PROGRAM SP1_2_Y111
VAR
	CompareOutput111_00: CMP_OC_DW;
	CompareOutput111_01: CMP_OC_DW;
	CompareOutput111_02: CMP_OC_DW;
	CompareOutput111_03: CMP_OC_DW;
	CompareOutput111_04: CMP_OC_DW;
	CompareOutput111_05: CMP_OC_DW;
	CompareOutput111_06: CMP_OC_DW;
	CompareOutput111_07: CMP_OC_DW;
	CompareOutput111_08: CMP_OC_DW;
	CompareOutput111_09: CMP_OC_DW;
	CompareOutput111_10: CMP_OC_DW;
	CompareOutput111_11: CMP_OC_DW;
	CompareOutput111_12: CMP_OC_DW;
	CompareOutput111_13: CMP_OC_DW;
	CompareOutput111_14: CMP_OC_DW;
	CompareOutput111_15: CMP_OC_DW;

END_VAR

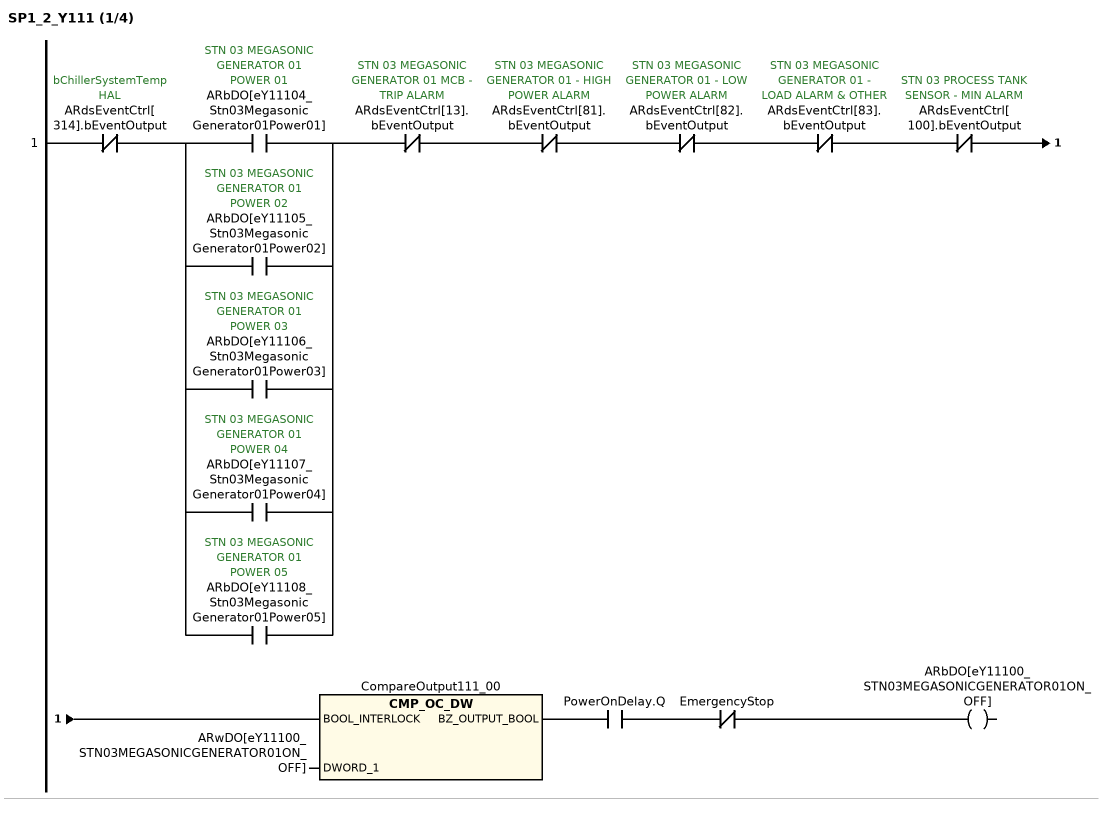
// NETWORK 1
//   ARdsEventCtrl[314].bEventOutput: bChillerSystemTempHAL
//   ARbDO[eY11104_Stn03MegasonicGenerator01Power01]: STN 03 MEGASONIC GENERATOR 01 POWER 01
//   ARbDO[eY11105_Stn03MegasonicGenerator01Power02]: STN 03 MEGASONIC GENERATOR 01 POWER 02
//   ARbDO[eY11106_Stn03MegasonicGenerator01Power03]: STN 03 MEGASONIC GENERATOR 01 POWER 03
//   ARbDO[eY11107_Stn03MegasonicGenerator01Power04]: STN 03 MEGASONIC GENERATOR 01 POWER 04
//   ARbDO[eY11108_Stn03MegasonicGenerator01Power05]: STN 03 MEGASONIC GENERATOR 01 POWER 05
//   ARdsEventCtrl[13].bEventOutput: STN 03 MEGASONIC GENERATOR 01 MCB - TRIP ALARM
//   ARdsEventCtrl[81].bEventOutput: STN 03 MEGASONIC GENERATOR 01 - HIGH POWER ALARM
//   ARdsEventCtrl[82].bEventOutput: STN 03 MEGASONIC GENERATOR 01 - LOW POWER ALARM
//   ARdsEventCtrl[83].bEventOutput: STN 03 MEGASONIC GENERATOR 01 - LOAD ALARM & OTHER
//   ARdsEventCtrl[100].bEventOutput: STN 03 PROCESS TANK SENSOR - MIN ALARM
CompareOutput111_00(BOOL_INTERLOCK := NOT ARdsEventCtrl[314].bEventOutput AND (ARbDO[eY11104_Stn03MegasonicGenerator01Power01] OR ARbDO[eY11105_Stn03MegasonicGenerator01Power02] OR ARbDO[eY11106_Stn03MegasonicGenerator01Power03] OR ARbDO[eY11107_Stn03MegasonicGenerator01Power04] OR ARbDO[eY11108_Stn03MegasonicGenerator01Power05]) AND NOT ARdsEventCtrl[13].bEventOutput AND NOT ARdsEventCtrl[81].bEventOutput AND NOT ARdsEventCtrl[82].bEventOutput AND NOT ARdsEventCtrl[83].bEventOutput AND NOT ARdsEventCtrl[100].bEventOutput, DWORD_1 := ARwDO[eY11100_STN03MEGASONICGENERATOR01ON_OFF]); // CMP_OC_DW
ARbDO[eY11100_STN03MEGASONICGENERATOR01ON_OFF] := CompareOutput111_00.BZ_OUTPUT_BOOL AND PowerOnDelay.Q AND NOT EmergencyStop;

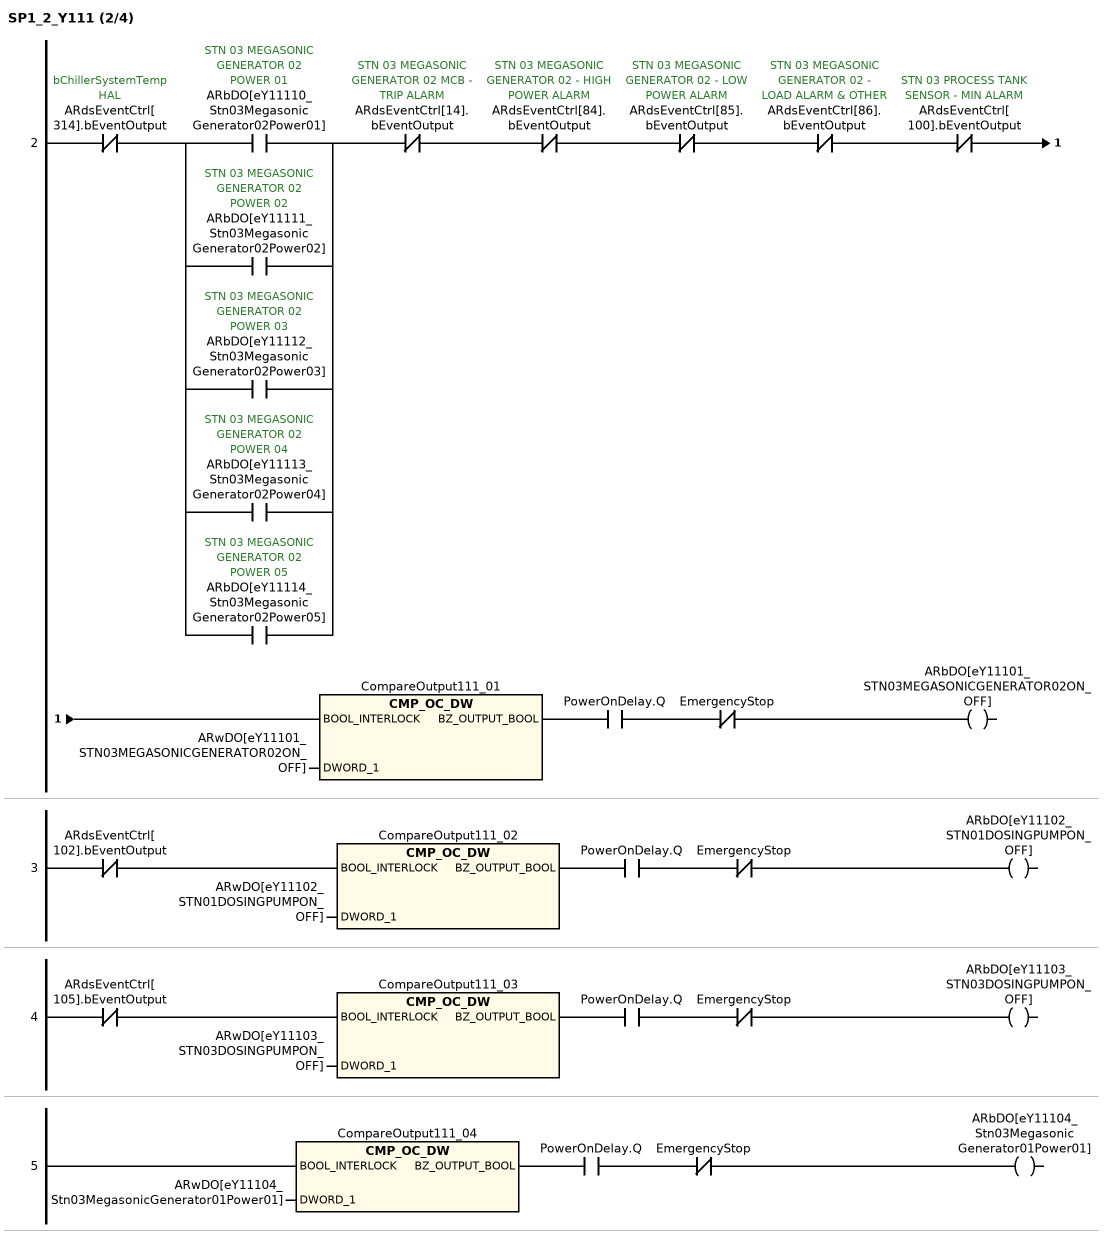
// NETWORK 2
//   ARdsEventCtrl[314].bEventOutput: bChillerSystemTempHAL
//   ARbDO[eY11110_Stn03MegasonicGenerator02Power01]: STN 03 MEGASONIC GENERATOR 02 POWER 01
//   ARbDO[eY11111_Stn03MegasonicGenerator02Power02]: STN 03 MEGASONIC GENERATOR 02 POWER 02
//   ARbDO[eY11112_Stn03MegasonicGenerator02Power03]: STN 03 MEGASONIC GENERATOR 02 POWER 03
//   ARbDO[eY11113_Stn03MegasonicGenerator02Power04]: STN 03 MEGASONIC GENERATOR 02 POWER 04
//   ARbDO[eY11114_Stn03MegasonicGenerator02Power05]: STN 03 MEGASONIC GENERATOR 02 POWER 05
//   ARdsEventCtrl[14].bEventOutput: STN 03 MEGASONIC GENERATOR 02 MCB - TRIP ALARM
//   ARdsEventCtrl[84].bEventOutput: STN 03 MEGASONIC GENERATOR 02 - HIGH POWER ALARM
//   ARdsEventCtrl[85].bEventOutput: STN 03 MEGASONIC GENERATOR 02 - LOW POWER ALARM
//   ARdsEventCtrl[86].bEventOutput: STN 03 MEGASONIC GENERATOR 02 - LOAD ALARM & OTHER
//   ARdsEventCtrl[100].bEventOutput: STN 03 PROCESS TANK SENSOR - MIN ALARM
CompareOutput111_01(BOOL_INTERLOCK := NOT ARdsEventCtrl[314].bEventOutput AND (ARbDO[eY11110_Stn03MegasonicGenerator02Power01] OR ARbDO[eY11111_Stn03MegasonicGenerator02Power02] OR ARbDO[eY11112_Stn03MegasonicGenerator02Power03] OR ARbDO[eY11113_Stn03MegasonicGenerator02Power04] OR ARbDO[eY11114_Stn03MegasonicGenerator02Power05]) AND NOT ARdsEventCtrl[14].bEventOutput AND NOT ARdsEventCtrl[84].bEventOutput AND NOT ARdsEventCtrl[85].bEventOutput AND NOT ARdsEventCtrl[86].bEventOutput AND NOT ARdsEventCtrl[100].bEventOutput, DWORD_1 := ARwDO[eY11101_STN03MEGASONICGENERATOR02ON_OFF]); // CMP_OC_DW
ARbDO[eY11101_STN03MEGASONICGENERATOR02ON_OFF] := CompareOutput111_01.BZ_OUTPUT_BOOL AND PowerOnDelay.Q AND NOT EmergencyStop;

// NETWORK 3
CompareOutput111_02(BOOL_INTERLOCK := NOT ARdsEventCtrl[102].bEventOutput, DWORD_1 := ARwDO[eY11102_STN01DOSINGPUMPON_OFF]); // CMP_OC_DW
ARbDO[eY11102_STN01DOSINGPUMPON_OFF] := CompareOutput111_02.BZ_OUTPUT_BOOL AND PowerOnDelay.Q AND NOT EmergencyStop;

// NETWORK 4
CompareOutput111_03(BOOL_INTERLOCK := NOT ARdsEventCtrl[105].bEventOutput, DWORD_1 := ARwDO[eY11103_STN03DOSINGPUMPON_OFF]); // CMP_OC_DW
ARbDO[eY11103_STN03DOSINGPUMPON_OFF] := CompareOutput111_03.BZ_OUTPUT_BOOL AND PowerOnDelay.Q AND NOT EmergencyStop;

// NETWORK 5
CompareOutput111_04(BOOL_INTERLOCK := TRUE, DWORD_1 := ARwDO[eY11104_Stn03MegasonicGenerator01Power01]); // CMP_OC_DW
ARbDO[eY11104_Stn03MegasonicGenerator01Power01] := CompareOutput111_04.BZ_OUTPUT_BOOL AND PowerOnDelay.Q AND NOT EmergencyStop;

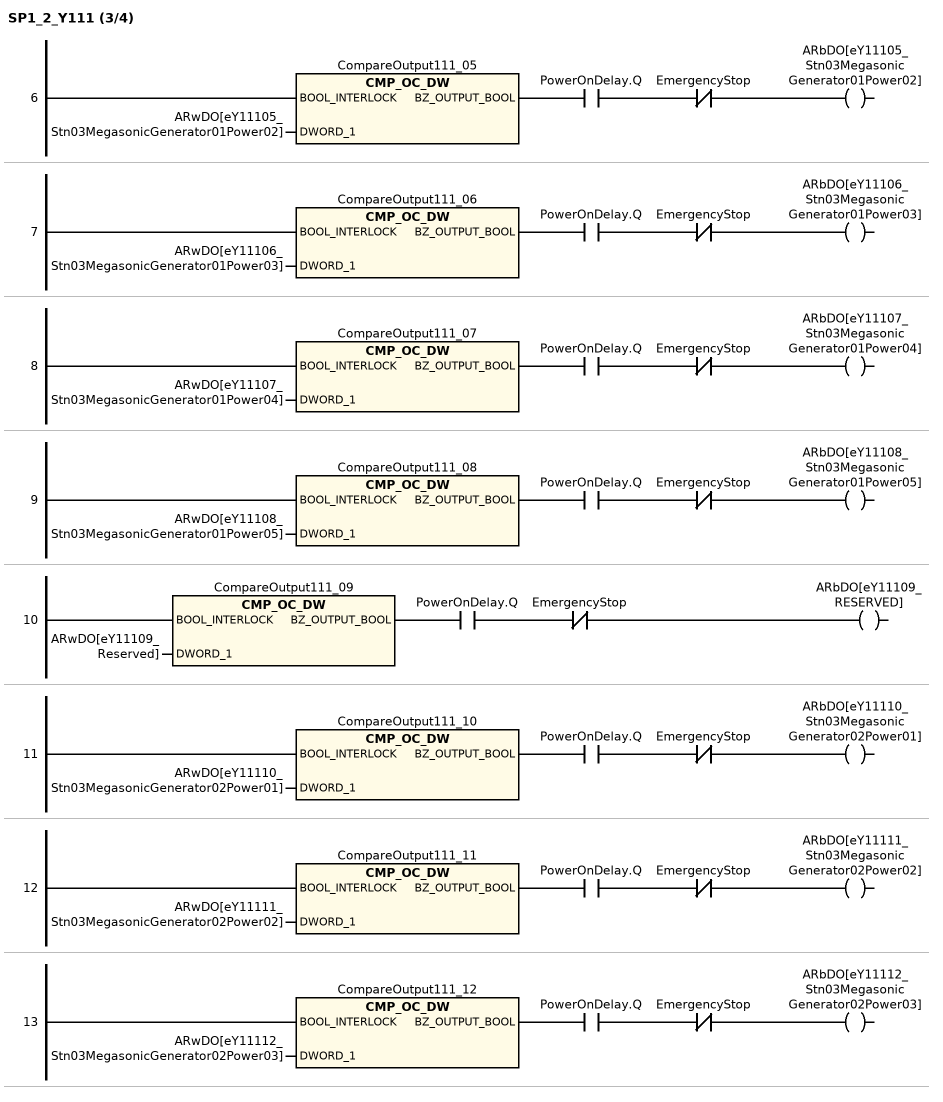
// NETWORK 6
CompareOutput111_05(BOOL_INTERLOCK := TRUE, DWORD_1 := ARwDO[eY11105_Stn03MegasonicGenerator01Power02]); // CMP_OC_DW
ARbDO[eY11105_Stn03MegasonicGenerator01Power02] := CompareOutput111_05.BZ_OUTPUT_BOOL AND PowerOnDelay.Q AND NOT EmergencyStop;

// NETWORK 7
CompareOutput111_06(BOOL_INTERLOCK := TRUE, DWORD_1 := ARwDO[eY11106_Stn03MegasonicGenerator01Power03]); // CMP_OC_DW
ARbDO[eY11106_Stn03MegasonicGenerator01Power03] := CompareOutput111_06.BZ_OUTPUT_BOOL AND PowerOnDelay.Q AND NOT EmergencyStop;

// NETWORK 8
CompareOutput111_07(BOOL_INTERLOCK := TRUE, DWORD_1 := ARwDO[eY11107_Stn03MegasonicGenerator01Power04]); // CMP_OC_DW
ARbDO[eY11107_Stn03MegasonicGenerator01Power04] := CompareOutput111_07.BZ_OUTPUT_BOOL AND PowerOnDelay.Q AND NOT EmergencyStop;

// NETWORK 9
CompareOutput111_08(BOOL_INTERLOCK := TRUE, DWORD_1 := ARwDO[eY11108_Stn03MegasonicGenerator01Power05]); // CMP_OC_DW
ARbDO[eY11108_Stn03MegasonicGenerator01Power05] := CompareOutput111_08.BZ_OUTPUT_BOOL AND PowerOnDelay.Q AND NOT EmergencyStop;

// NETWORK 10
CompareOutput111_09(BOOL_INTERLOCK := TRUE, DWORD_1 := ARwDO[eY11109_Reserved]); // CMP_OC_DW
ARbDO[eY11109_RESERVED] := CompareOutput111_09.BZ_OUTPUT_BOOL AND PowerOnDelay.Q AND NOT EmergencyStop;

// NETWORK 11
CompareOutput111_10(BOOL_INTERLOCK := TRUE, DWORD_1 := ARwDO[eY11110_Stn03MegasonicGenerator02Power01]); // CMP_OC_DW
ARbDO[eY11110_Stn03MegasonicGenerator02Power01] := CompareOutput111_10.BZ_OUTPUT_BOOL AND PowerOnDelay.Q AND NOT EmergencyStop;

// NETWORK 12
CompareOutput111_11(BOOL_INTERLOCK := TRUE, DWORD_1 := ARwDO[eY11111_Stn03MegasonicGenerator02Power02]); // CMP_OC_DW
ARbDO[eY11111_Stn03MegasonicGenerator02Power02] := CompareOutput111_11.BZ_OUTPUT_BOOL AND PowerOnDelay.Q AND NOT EmergencyStop;

// NETWORK 13
CompareOutput111_12(BOOL_INTERLOCK := TRUE, DWORD_1 := ARwDO[eY11112_Stn03MegasonicGenerator02Power03]); // CMP_OC_DW
ARbDO[eY11112_Stn03MegasonicGenerator02Power03] := CompareOutput111_12.BZ_OUTPUT_BOOL AND PowerOnDelay.Q AND NOT EmergencyStop;

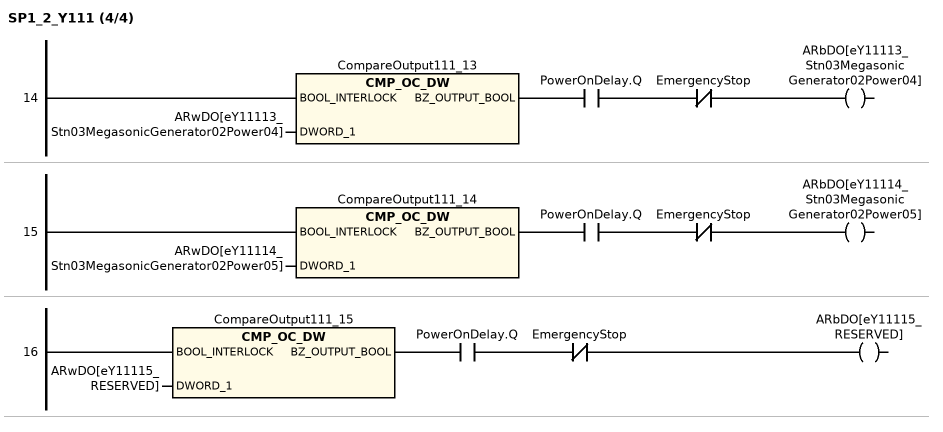
// NETWORK 14
CompareOutput111_13(BOOL_INTERLOCK := TRUE, DWORD_1 := ARwDO[eY11113_Stn03MegasonicGenerator02Power04]); // CMP_OC_DW
ARbDO[eY11113_Stn03MegasonicGenerator02Power04] := CompareOutput111_13.BZ_OUTPUT_BOOL AND PowerOnDelay.Q AND NOT EmergencyStop;

// NETWORK 15
CompareOutput111_14(BOOL_INTERLOCK := TRUE, DWORD_1 := ARwDO[eY11114_Stn03MegasonicGenerator02Power05]); // CMP_OC_DW
ARbDO[eY11114_Stn03MegasonicGenerator02Power05] := CompareOutput111_14.BZ_OUTPUT_BOOL AND PowerOnDelay.Q AND NOT EmergencyStop;

// NETWORK 16
CompareOutput111_15(BOOL_INTERLOCK := TRUE, DWORD_1 := ARwDO[eY11115_RESERVED]); // CMP_OC_DW
ARbDO[eY11115_RESERVED] := CompareOutput111_15.BZ_OUTPUT_BOOL AND PowerOnDelay.Q AND NOT EmergencyStop;

END_PROGRAM

(* stored: Version 1.1.0.1, ProductVersion 3.1.4024.11
   POU SP1_2_Y111: Id {db4ecc1b-2b14-445b-8a42-d2e300fdc819}, SpecialFunc None *)
